{attribute 'GeneratedUsingTerminal: EK1122-0000-0018'}
{attribute addProperty BoxType "EK1122-0000-0018"}
{attribute addProperty Id "Beckhoff_EL5xxxsub_EK1100EK1100_1FC0878B2"}
{attribute addProperty CRC "1829247018"}
{attribute addProperty Size "2"}
TYPE Beckhoff_EL5xxxEK1122_6D08182A EXTENDS EK1122_1FC0878B :
STRUCT
	{attribute addProperty Name "Beckhoff_EL5xxxsub_EK1100"}
	{attribute addProperty PreviousPort "Beckhoff EL5xxxEK1122 : D"}
	Beckhoff_EL5xxxsub_EK1100 : EK1100_1FC0878B;
END_STRUCT
END_TYPE

(* stored: Version 1.2.0.0, ProductVersion 3.1.4024.9
   DUT Beckhoff_EL5xxxEK1122_6D08182A: Id {68ad389c-7782-47b0-8997-44265322c14e} *)
